GLOBALCONSTANTS quarterconst (* Global constants *)
  (* Standard: 61499-1 *)
  (* Version 1.0, 2024-02-22, franz *)
  VAR_GLOBAL CONSTANT
    BYTE_QUARTER_ZZ : BYTE := 2#0000_0000; (* ZERO Constant *)
    SHIFT_QUARTER_00 : SINT := 0; (* shift 0 bits *)
    BYTE_QUARTER_00 : BYTE := 2#0000_0011; (* quarter byte 00 Constant *)
    SHIFT_QUARTER_01 : SINT := 2; (* shift 2 bits *)
    BYTE_QUARTER_01 : BYTE := 2#0000_1100; (* quarter byte 01 Constant *)
    SHIFT_QUARTER_02 : SINT := 4; (* shift 4 bits *)
    BYTE_QUARTER_02 : BYTE := 2#0011_0000; (* quarter byte 02 Constant *)
    SHIFT_QUARTER_03 : SINT := 6; (* shift 6 bits *)
    BYTE_QUARTER_03 : BYTE := 2#1100_0000; (* quarter byte 03 Constant *)
    WORD_QUARTER_ZZ : WORD := 2#0000_0000_0000_0000; (* ZERO Constant *)
    WORD_QUARTER_00 : WORD := 2#0000_0000_0000_0011; (* quarter WORD 00 Constant *)
    WORD_QUARTER_01 : WORD := 2#0000_0000_0000_1100; (* quarter WORD 01 Constant *)
    WORD_QUARTER_02 : WORD := 2#0000_0000_0011_0000; (* quarter WORD 02 Constant *)
    WORD_QUARTER_03 : WORD := 2#0000_0000_1100_0000; (* quarter WORD 03 Constant *)
    SHIFT_QUARTER_04 : SINT := 8; (* shift 8 bits *)
    WORD_QUARTER_04 : WORD := 2#0000_0011_0000_0000; (* quarter WORD 04 Constant *)
    SHIFT_QUARTER_05 : SINT := 10; (* shift 10 bits *)
    WORD_QUARTER_05 : WORD := 2#0000_1100_0000_0000; (* quarter WORD 05 Constant *)
    SHIFT_QUARTER_06 : SINT := 12; (* shift 12 bits *)
    WORD_QUARTER_06 : WORD := 2#0011_0000_0000_0000; (* quarter WORD 06 Constant *)
    SHIFT_QUARTER_07 : SINT := 14; (* shift 14 bits *)
    WORD_QUARTER_07 : WORD := 2#1100_0000_0000_0000; (* quarter WORD 07 Constant *)
    DWORD_QUARTER_ZZ : DWORD := 2#0000_0000_0000_0000_0000_0000_0000_0000; (* ZERO Constant *)
    DWORD_QUARTER_00 : DWORD := 2#0000_0000_0000_0000_0000_0000_0000_0011; (* quarter DWORD 00 Constant *)
    DWORD_QUARTER_01 : DWORD := 2#0000_0000_0000_0000_0000_0000_0000_1100; (* quarter DWORD 01 Constant *)
    DWORD_QUARTER_02 : DWORD := 2#0000_0000_0000_0000_0000_0000_0011_0000; (* quarter DWORD 02 Constant *)
    DWORD_QUARTER_03 : DWORD := 2#0000_0000_0000_0000_0000_0000_1100_0000; (* quarter DWORD 03 Constant *)
    DWORD_QUARTER_04 : DWORD := 2#0000_0000_0000_0000_0000_0011_0000_0000; (* quarter DWORD 04 Constant *)
    DWORD_QUARTER_05 : DWORD := 2#0000_0000_0000_0000_0000_1100_0000_0000; (* quarter DWORD 05 Constant *)
    DWORD_QUARTER_06 : DWORD := 2#0000_0000_0000_0000_0011_0000_0000_0000; (* quarter DWORD 06 Constant *)
    DWORD_QUARTER_07 : DWORD := 2#0000_0000_0000_0000_1100_0000_0000_0000; (* quarter DWORD 07 Constant *)
    SHIFT_QUARTER_08 : SINT := 16; (* shift 16 bits *)
    DWORD_QUARTER_08 : DWORD := 2#0000_0000_0000_0011_0000_0000_0000_0000; (* quarter DWORD 08 Constant *)
    SHIFT_QUARTER_09 : SINT := 18; (* shift 18 bits *)
    DWORD_QUARTER_09 : DWORD := 2#0000_0000_0000_1100_0000_0000_0000_0000; (* quarter DWORD 09 Constant *)
    SHIFT_QUARTER_10 : SINT := 20; (* shift 20 bits *)
    DWORD_QUARTER_10 : DWORD := 2#0000_0000_0011_0000_0000_0000_0000_0000; (* quarter DWORD 10 Constant *)
    SHIFT_QUARTER_11 : SINT := 22; (* shift 22 bits *)
    DWORD_QUARTER_11 : DWORD := 2#0000_0000_1100_0000_0000_0000_0000_0000; (* quarter DWORD 11 Constant *)
    SHIFT_QUARTER_12 : SINT := 24; (* shift 24 bits *)
    DWORD_QUARTER_12 : DWORD := 2#0000_0011_0000_0000_0000_0000_0000_0000; (* quarter DWORD 12 Constant *)
    SHIFT_QUARTER_13 : SINT := 26; (* shift 26 bits *)
    DWORD_QUARTER_13 : DWORD := 2#0000_1100_0000_0000_0000_0000_0000_0000; (* quarter DWORD 13 Constant *)
    SHIFT_QUARTER_14 : SINT := 28; (* shift 28 bits *)
    DWORD_QUARTER_14 : DWORD := 2#0011_0000_0000_0000_0000_0000_0000_0000; (* quarter DWORD 14 Constant *)
    SHIFT_QUARTER_15 : SINT := 30; (* shift 30 bits *)
    DWORD_QUARTER_15 : DWORD := 2#1100_0000_0000_0000_0000_0000_0000_0000; (* quarter DWORD 15 Constant *)
    LWORD_QUARTER_ZZ : LWORD := 2#0000_0000_0000_0000_0000_0000_0000_0000_0000_0000_0000_0000_0000_0000_0000_0000; (* ZERO Constant *)
    LWORD_QUARTER_00 : LWORD := 2#0000_0000_0000_0000_0000_0000_0000_0000_0000_0000_0000_0000_0000_0000_0000_0011; (* quarter LWORD 00 Constant *)
    LWORD_QUARTER_01 : LWORD := 2#0000_0000_0000_0000_0000_0000_0000_0000_0000_0000_0000_0000_0000_0000_0000_1100; (* quarter LWORD 01 Constant *)
    LWORD_QUARTER_02 : LWORD := 2#0000_0000_0000_0000_0000_0000_0000_0000_0000_0000_0000_0000_0000_0000_0011_0000; (* quarter LWORD 02 Constant *)
    LWORD_QUARTER_03 : LWORD := 2#0000_0000_0000_0000_0000_0000_0000_0000_0000_0000_0000_0000_0000_0000_1100_0000; (* quarter LWORD 03 Constant *)
    LWORD_QUARTER_04 : LWORD := 2#0000_0000_0000_0000_0000_0000_0000_0000_0000_0000_0000_0000_0000_0011_0000_0000; (* quarter LWORD 04 Constant *)
    LWORD_QUARTER_05 : LWORD := 2#0000_0000_0000_0000_0000_0000_0000_0000_0000_0000_0000_0000_0000_1100_0000_0000; (* quarter LWORD 05 Constant *)
    LWORD_QUARTER_06 : LWORD := 2#0000_0000_0000_0000_0000_0000_0000_0000_0000_0000_0000_0000_0011_0000_0000_0000; (* quarter LWORD 06 Constant *)
    LWORD_QUARTER_07 : LWORD := 2#0000_0000_0000_0000_0000_0000_0000_0000_0000_0000_0000_0000_1100_0000_0000_0000; (* quarter LWORD 07 Constant *)
    LWORD_QUARTER_08 : LWORD := 2#0000_0000_0000_0000_0000_0000_0000_0000_0000_0000_0000_0011_0000_0000_0000_0000; (* quarter LWORD 08 Constant *)
    LWORD_QUARTER_09 : LWORD := 2#0000_0000_0000_0000_0000_0000_0000_0000_0000_0000_0000_1100_0000_0000_0000_0000; (* quarter LWORD 09 Constant *)
    LWORD_QUARTER_10 : LWORD := 2#0000_0000_0000_0000_0000_0000_0000_0000_0000_0000_0011_0000_0000_0000_0000_0000; (* quarter LWORD 10 Constant *)
    LWORD_QUARTER_11 : LWORD := 2#0000_0000_0000_0000_0000_0000_0000_0000_0000_0000_1100_0000_0000_0000_0000_0000; (* quarter LWORD 11 Constant *)
    LWORD_QUARTER_12 : LWORD := 2#0000_0000_0000_0000_0000_0000_0000_0000_0000_0011_0000_0000_0000_0000_0000_0000; (* quarter LWORD 12 Constant *)
    LWORD_QUARTER_13 : LWORD := 2#0000_0000_0000_0000_0000_0000_0000_0000_0000_1100_0000_0000_0000_0000_0000_0000; (* quarter LWORD 13 Constant *)
    LWORD_QUARTER_14 : LWORD := 2#0000_0000_0000_0000_0000_0000_0000_0000_0011_0000_0000_0000_0000_0000_0000_0000; (* quarter LWORD 14 Constant *)
    LWORD_QUARTER_15 : LWORD := 2#0000_0000_0000_0000_0000_0000_0000_0000_1100_0000_0000_0000_0000_0000_0000_0000; (* quarter LWORD 15 Constant *)
    SHIFT_QUARTER_16 : SINT := 32; (* shift 32 bits *)
    LWORD_QUARTER_16 : LWORD := 2#0000_0000_0000_0000_0000_0000_0000_0011_0000_0000_0000_0000_0000_0000_0000_0000; (* quarter LWORD 16 Constant *)
    SHIFT_QUARTER_17 : SINT := 34; (* shift 34 bits *)
    LWORD_QUARTER_17 : LWORD := 2#0000_0000_0000_0000_0000_0000_0000_1100_0000_0000_0000_0000_0000_0000_0000_0000; (* quarter LWORD 17 Constant *)
    SHIFT_QUARTER_18 : SINT := 36; (* shift 36 bits *)
    LWORD_QUARTER_18 : LWORD := 2#0000_0000_0000_0000_0000_0000_0011_0000_0000_0000_0000_0000_0000_0000_0000_0000; (* quarter LWORD 18 Constant *)
    SHIFT_QUARTER_19 : SINT := 38; (* shift 38 bits *)
    LWORD_QUARTER_19 : LWORD := 2#0000_0000_0000_0000_0000_0000_1100_0000_0000_0000_0000_0000_0000_0000_0000_0000; (* quarter LWORD 19 Constant *)
    SHIFT_QUARTER_20 : SINT := 40; (* shift 40 bits *)
    LWORD_QUARTER_20 : LWORD := 2#0000_0000_0000_0000_0000_0011_0000_0000_0000_0000_0000_0000_0000_0000_0000_0000; (* quarter LWORD 20 Constant *)
    SHIFT_QUARTER_21 : SINT := 42; (* shift 42 bits *)
    LWORD_QUARTER_21 : LWORD := 2#0000_0000_0000_0000_0000_1100_0000_0000_0000_0000_0000_0000_0000_0000_0000_0000; (* quarter LWORD 21 Constant *)
    SHIFT_QUARTER_22 : SINT := 44; (* shift 44 bits *)
    LWORD_QUARTER_22 : LWORD := 2#0000_0000_0000_0000_0011_0000_0000_0000_0000_0000_0000_0000_0000_0000_0000_0000; (* quarter LWORD 22 Constant *)
    SHIFT_QUARTER_23 : SINT := 46; (* shift 46 bits *)
    LWORD_QUARTER_23 : LWORD := 2#0000_0000_0000_0000_1100_0000_0000_0000_0000_0000_0000_0000_0000_0000_0000_0000; (* quarter LWORD 23 Constant *)
    SHIFT_QUARTER_24 : SINT := 48; (* shift 48 bits *)
    LWORD_QUARTER_24 : LWORD := 2#0000_0000_0000_0011_0000_0000_0000_0000_0000_0000_0000_0000_0000_0000_0000_0000; (* quarter LWORD 24 Constant *)
    SHIFT_QUARTER_25 : SINT := 50; (* shift 50 bits *)
    LWORD_QUARTER_25 : LWORD := 2#0000_0000_0000_1100_0000_0000_0000_0000_0000_0000_0000_0000_0000_0000_0000_0000; (* quarter LWORD 25 Constant *)
    SHIFT_QUARTER_26 : SINT := 52; (* shift 52 bits *)
    LWORD_QUARTER_26 : LWORD := 2#0000_0000_0011_0000_0000_0000_0000_0000_0000_0000_0000_0000_0000_0000_0000_0000; (* quarter LWORD 26 Constant *)
    SHIFT_QUARTER_27 : SINT := 54; (* shift 54 bits *)
    LWORD_QUARTER_27 : LWORD := 2#0000_0000_1100_0000_0000_0000_0000_0000_0000_0000_0000_0000_0000_0000_0000_0000; (* quarter LWORD 27 Constant *)
    SHIFT_QUARTER_28 : SINT := 56; (* shift 56 bits *)
    LWORD_QUARTER_28 : LWORD := 2#0000_0011_0000_0000_0000_0000_0000_0000_0000_0000_0000_0000_0000_0000_0000_0000; (* quarter LWORD 28 Constant *)
    SHIFT_QUARTER_29 : SINT := 58; (* shift 58 bits *)
    LWORD_QUARTER_29 : LWORD := 2#0000_1100_0000_0000_0000_0000_0000_0000_0000_0000_0000_0000_0000_0000_0000_0000; (* quarter LWORD 29 Constant *)
    SHIFT_QUARTER_30 : SINT := 60; (* shift 60 bits *)
    LWORD_QUARTER_30 : LWORD := 2#0011_0000_0000_0000_0000_0000_0000_0000_0000_0000_0000_0000_0000_0000_0000_0000; (* quarter LWORD 30 Constant *)
    SHIFT_QUARTER_31 : SINT := 62; (* shift 62 bits *)
    LWORD_QUARTER_31 : LWORD := 2#1100_0000_0000_0000_0000_0000_0000_0000_0000_0000_0000_0000_0000_0000_0000_0000; (* quarter LWORD 31 Constant *)
  END_VAR
END_GLOBALCONSTANTS
